PROGRAM MAIN
VAR PERSISTENT
	SW_Liste:SW_Struct;
END_VAR
VAR
	VD_0: VD;
	Kreis_3KO_0: Kreis_3KO;
	KD_0: KD;
	IOs_0: IOs;
	AI_to_Druck_0: AI_to_Druck;
	AI_to_Druck_1: AI_to_Druck;
	Init_0: Init;
	i_anzahlStufen: INT;
	einestufe: BOOL;
	zweitestufe: BOOL;
	Logger_0: logger;
	COUNT_0: count;
END_VAR

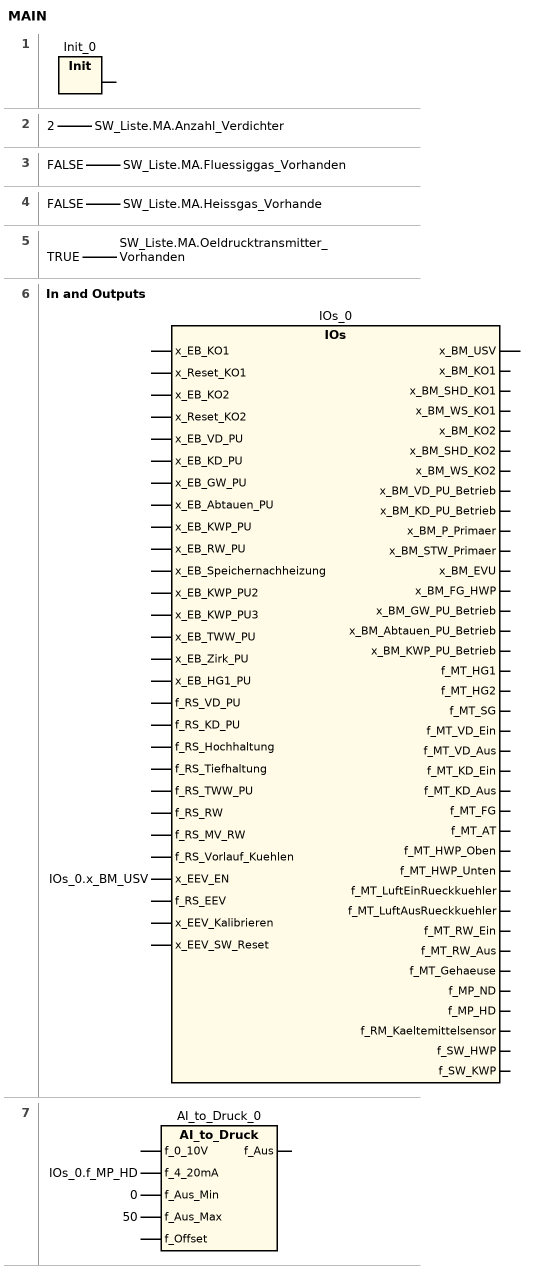
// NETWORK 1
Init_0(); // Init

// NETWORK 2
SW_Liste.MA.Anzahl_Verdichter := 2;

// NETWORK 3
SW_Liste.MA.Fluessiggas_Vorhanden := FALSE;

// NETWORK 4
SW_Liste.MA.Heissgas_Vorhande := FALSE;

// NETWORK 5
SW_Liste.MA.Oeldrucktransmitter_Vorhanden := TRUE;

// NETWORK 6: In and Outputs
IOs_0(x_EEV_EN := IOs_0.x_BM_USV); // IOs

// NETWORK 7
AI_to_Druck_0(f_4_20mA := IOs_0.f_MP_HD, f_Aus_Min := 0, f_Aus_Max := 50); // AI_to_Druck

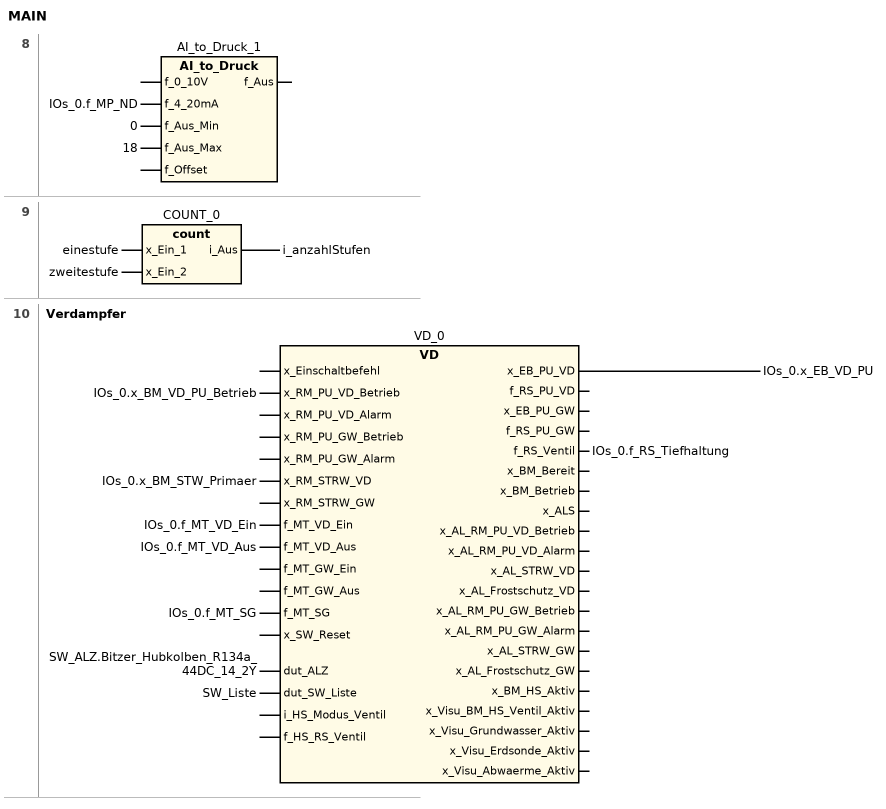
// NETWORK 8
AI_to_Druck_1(f_4_20mA := IOs_0.f_MP_ND, f_Aus_Min := 0, f_Aus_Max := 18); // AI_to_Druck

// NETWORK 9
COUNT_0(x_Ein_1 := einestufe, x_Ein_2 := zweitestufe); // count
i_anzahlStufen := COUNT_0.i_Aus;

// NETWORK 10: Verdampfer
VD_0(
    x_RM_PU_VD_Betrieb := IOs_0.x_BM_VD_PU_Betrieb,
    x_RM_STRW_VD := IOs_0.x_BM_STW_Primaer,
    f_MT_VD_Ein := IOs_0.f_MT_VD_Ein,
    f_MT_VD_Aus := IOs_0.f_MT_VD_Aus,
    f_MT_SG := IOs_0.f_MT_SG,
    dut_ALZ := SW_ALZ.Bitzer_Hubkolben_R134a_44DC_14_2Y,
    dut_SW_Liste := SW_Liste,
    f_RS_Ventil => IOs_0.f_RS_Tiefhaltung); // VD
IOs_0.x_EB_VD_PU := VD_0.x_EB_PU_VD;

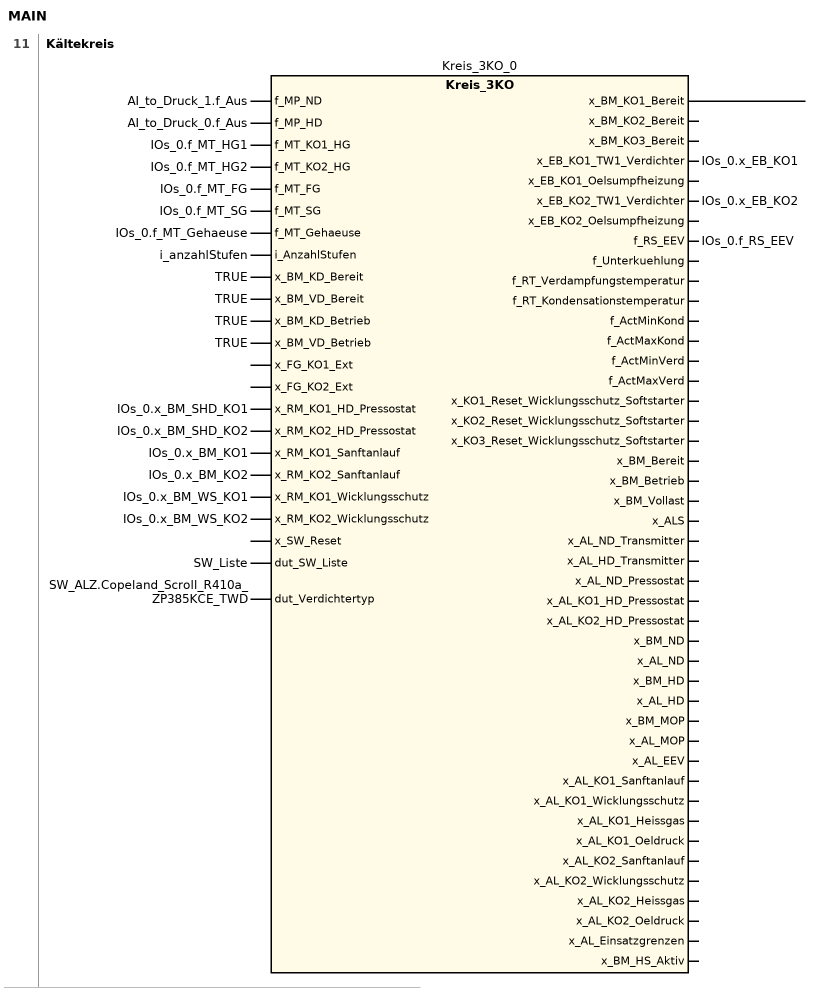
// NETWORK 11: Kältekreis
Kreis_3KO_0(
    f_MP_ND := AI_to_Druck_1.f_Aus,
    f_MP_HD := AI_to_Druck_0.f_Aus,
    f_MT_KO1_HG := IOs_0.f_MT_HG1,
    f_MT_KO2_HG := IOs_0.f_MT_HG2,
    f_MT_FG := IOs_0.f_MT_FG,
    f_MT_SG := IOs_0.f_MT_SG,
    f_MT_Gehaeuse := IOs_0.f_MT_Gehaeuse,
    i_AnzahlStufen := i_anzahlStufen,
    x_BM_KD_Bereit := TRUE,
    x_BM_VD_Bereit := TRUE,
    x_BM_KD_Betrieb := TRUE,
    x_BM_VD_Betrieb := TRUE,
    x_RM_KO1_HD_Pressostat := IOs_0.x_BM_SHD_KO1,
    x_RM_KO2_HD_Pressostat := IOs_0.x_BM_SHD_KO2,
    x_RM_KO1_Sanftanlauf := IOs_0.x_BM_KO1,
    x_RM_KO2_Sanftanlauf := IOs_0.x_BM_KO2,
    x_RM_KO1_Wicklungsschutz := IOs_0.x_BM_WS_KO1,
    x_RM_KO2_Wicklungsschutz := IOs_0.x_BM_WS_KO2,
    dut_SW_Liste := SW_Liste,
    dut_Verdichtertyp := SW_ALZ.Copeland_Scroll_R410a_ZP385KCE_TWD,
    x_EB_KO1_TW1_Verdichter => IOs_0.x_EB_KO1,
    x_EB_KO2_TW1_Verdichter => IOs_0.x_EB_KO2,
    f_RS_EEV => IOs_0.f_RS_EEV); // Kreis_3KO

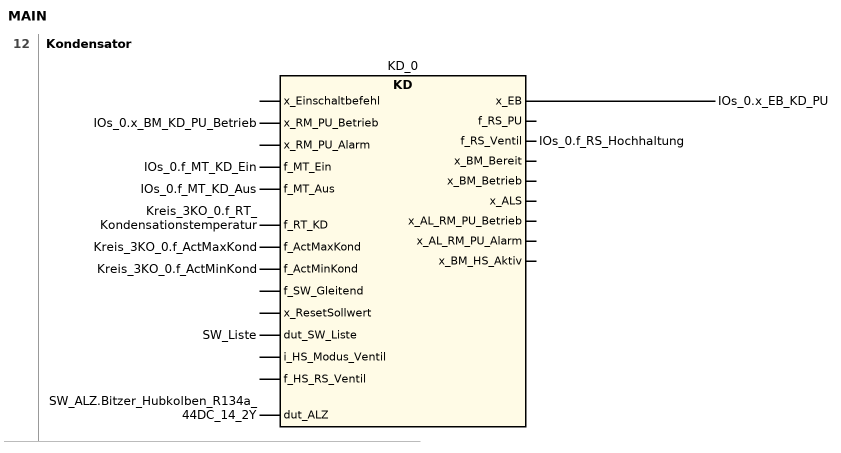
// NETWORK 12: Kondensator
KD_0(
    x_RM_PU_Betrieb := IOs_0.x_BM_KD_PU_Betrieb,
    f_MT_Ein := IOs_0.f_MT_KD_Ein,
    f_MT_Aus := IOs_0.f_MT_KD_Aus,
    f_RT_KD := Kreis_3KO_0.f_RT_Kondensationstemperatur,
    f_ActMaxKond := Kreis_3KO_0.f_ActMaxKond,
    f_ActMinKond := Kreis_3KO_0.f_ActMinKond,
    dut_SW_Liste := SW_Liste,
    dut_ALZ := SW_ALZ.Bitzer_Hubkolben_R134a_44DC_14_2Y,
    f_RS_Ventil => IOs_0.f_RS_Hochhaltung); // KD
IOs_0.x_EB_KD_PU := KD_0.x_EB;

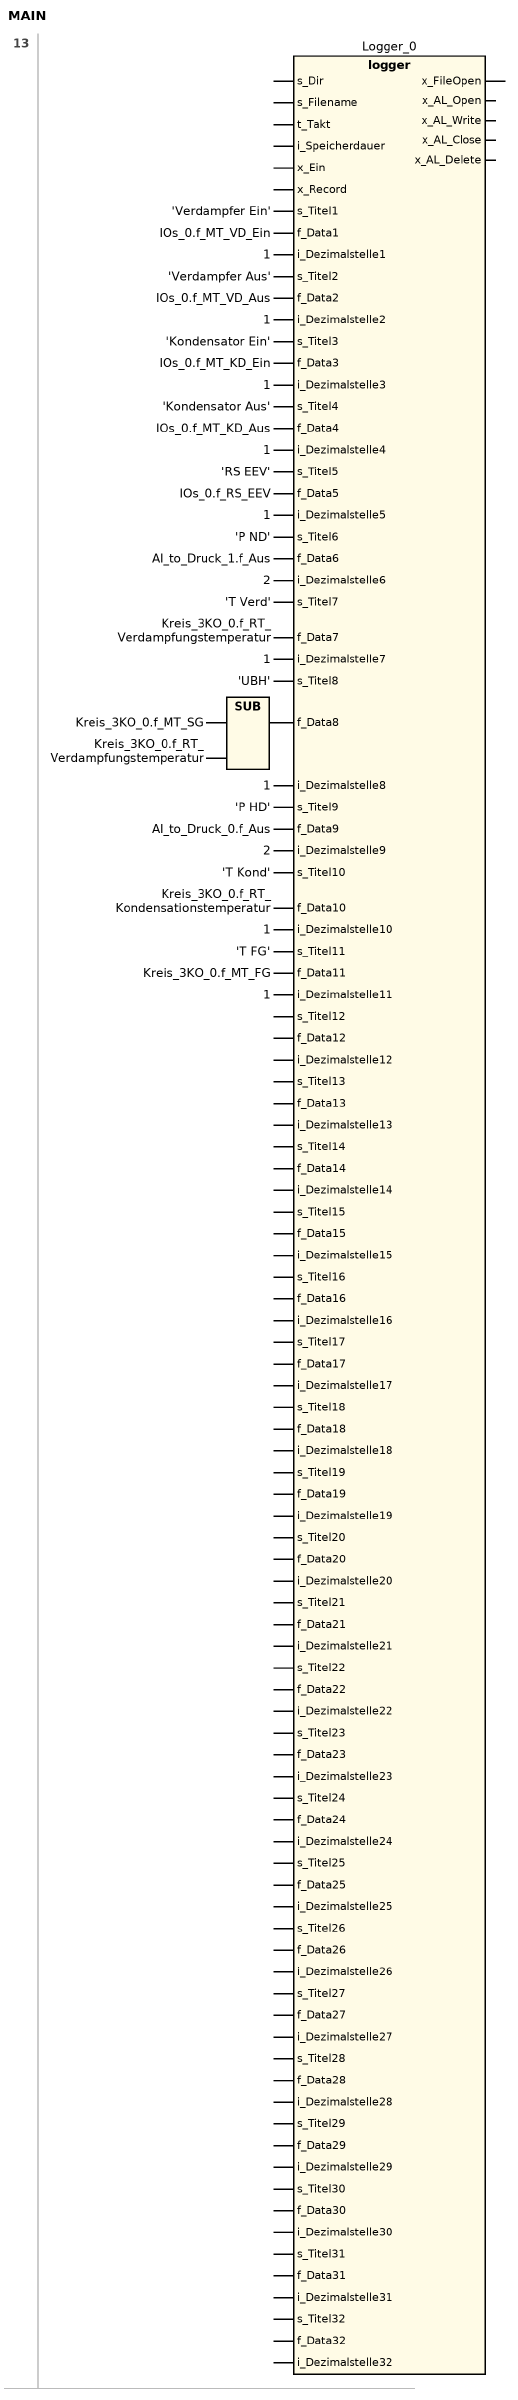
// NETWORK 13
Logger_0(
    s_Titel1 := 'Verdampfer Ein',
    f_Data1 := IOs_0.f_MT_VD_Ein,
    i_Dezimalstelle1 := 1,
    s_Titel2 := 'Verdampfer Aus',
    f_Data2 := IOs_0.f_MT_VD_Aus,
    i_Dezimalstelle2 := 1,
    s_Titel3 := 'Kondensator Ein',
    f_Data3 := IOs_0.f_MT_KD_Ein,
    i_Dezimalstelle3 := 1,
    s_Titel4 := 'Kondensator Aus',
    f_Data4 := IOs_0.f_MT_KD_Aus,
    i_Dezimalstelle4 := 1,
    s_Titel5 := 'RS EEV',
    f_Data5 := IOs_0.f_RS_EEV,
    i_Dezimalstelle5 := 1,
    s_Titel6 := 'P ND',
    f_Data6 := AI_to_Druck_1.f_Aus,
    i_Dezimalstelle6 := 2,
    s_Titel7 := 'T Verd',
    f_Data7 := Kreis_3KO_0.f_RT_Verdampfungstemperatur,
    i_Dezimalstelle7 := 1,
    s_Titel8 := 'UBH',
    f_Data8 := Kreis_3KO_0.f_MT_SG - Kreis_3KO_0.f_RT_Verdampfungstemperatur,
    i_Dezimalstelle8 := 1,
    s_Titel9 := 'P HD',
    f_Data9 := AI_to_Druck_0.f_Aus,
    i_Dezimalstelle9 := 2,
    s_Titel10 := 'T Kond',
    f_Data10 := Kreis_3KO_0.f_RT_Kondensationstemperatur,
    i_Dezimalstelle10 := 1,
    s_Titel11 := 'T FG',
    f_Data11 := Kreis_3KO_0.f_MT_FG,
    i_Dezimalstelle11 := 1); // logger

END_PROGRAM

(* stored: Version 1.1.0.1, ProductVersion 3.1.4022.6
   POU MAIN: Id {3eff947f-98b6-4c36-8068-08914cf48de2}, SpecialFunc None *)
